// Mitsubishi GX Works2 project: z02   PLC: Q02/Q02H

PROGRAM MAIN
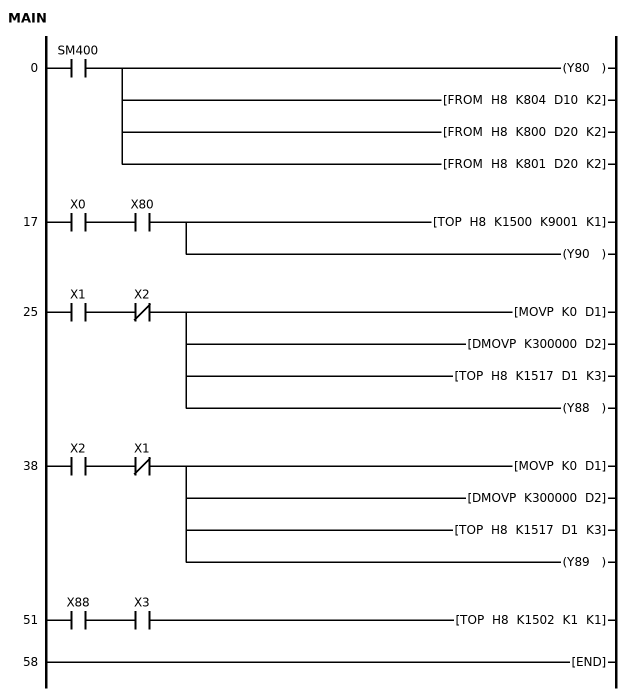
0     LD      SM400
      OUT     Y80
      FROM    H8 K804 D10 K2
      FROM    H8 K800 D20 K2
      FROM    H8 K801 D20 K2
17    LD      X0
      AND     X80
      TOP     H8 K1500 K9001 K1
      OUT     Y90
25    LD      X1
      ANI     X2
      MOVP    K0 D1
      DMOVP   K300000 D2
      TOP     H8 K1517 D1 K3
      OUT     Y88
38    LD      X2
      ANI     X1
      MOVP    K0 D1
      DMOVP   K300000 D2
      TOP     H8 K1517 D1 K3
      OUT     Y89
51    LD      X88
      AND     X3
      TOP     H8 K1502 K1 K1
58    END
END_PROGRAM
